Yaskawa INFORM job: CUTPKT.JBI

/JOB
//NAME CUTPKT
//POS
///NPOS 1,1,1,0,0,0
///TOOL 29
///POSTYPE PULSE
///PULSE
C00000=10645,-114998,-116552,5579,58952,90735
///TOOL 0
BC00000=204899,680330,1075141
EC00000=798153,1112947
//INST
///DATE 2024/01/11 10:27
///ATTR SC,RW
///GROUP1 RB1,BS1
///GROUP2 ST1
NOP
MOVJ C00000 BC00000 VJ=0.78  +MOVJ EC00000 VJ=0.78
END
